Universal Robots PolyScope program: speedSliderEx_wInput.urp

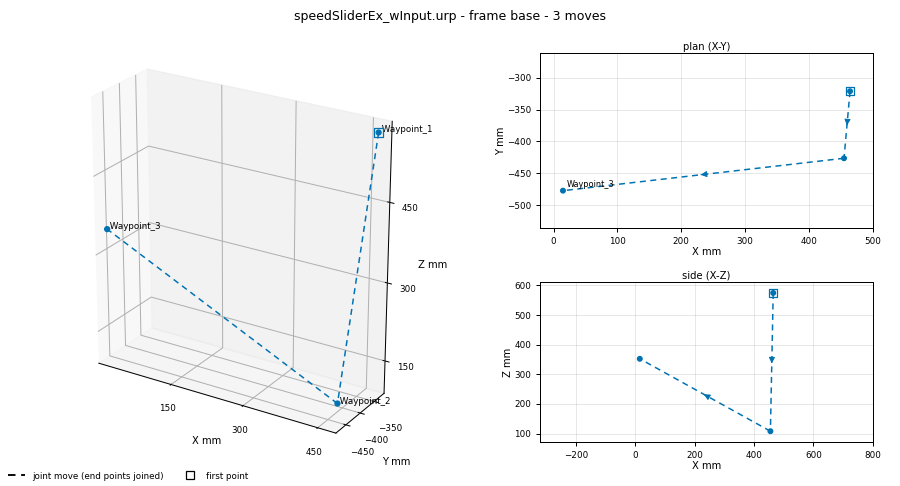
[picture p0: tool path of speedSliderEx_wInput.urp in frame base, 3 of 3 moves have a stored position in this frame; points joined in program order, loops and branches not executed]
ProgramRoot directory=/programs; kinematics=(a=[0, -0.425, -0.39225, 0, 0, 0], d=[0.08916, 0, 0, 0.10915, 0.09465, 0.0823], alpha=[1.5708, 0, 0, 1.5708, -1.5708, 0], deltaTheta=[0, 0, 0, 0, 0, 0], status=notInitialized); name=speedSliderEx_wInput; programVersion=(project__name=PolyScope, major__version=1, minor__version=8, svn__revision=14035, build__date=Apr 28 2014, 10:06:36); robotEnvironmentFileName=default; serialNumberRobot=2012209394
  MainProgram cartesianAcceleration=1.2; cartesianSpeed=12.0; jointAcceleration=1.3962634015954636; jointSpeed=1.0471975511965976; moveAsFastAsPossible=true; sharedProcessMoveBlendRadius=0.025; featureReference=(installationNameReference=Base); motionType=JOINT_SPACE
    Move cartesianAcceleration=1.2; cartesianSpeed=12.0; jointAcceleration=1.3962634015954636; jointSpeed=1.0471975511965976; moveAsFastAsPossible=true; sharedProcessMoveBlendRadius=0.025; featureReference=(installationNameReference=Base); motionType=JOINT_SPACE
      Waypoint blendRadius=0.05; cartesianAcceleration=1.2; cartesianSpeed=12.0; jointAcceleration=1.3962634015954636; jointSpeed=1.0471975511965976; nextMotionTime=2.0; stoppoint=true; useSharedBlendParameter=true; useSharedParameters=true; position=TCP in base x=464.486 y=-321.339 z=574.383 mm, rx=2.3556 ry=2.0077 rz=0.0323 rad; joints [-23.52, -102.508, -55.368, -109.215, 89.91, -194.406] deg; positionType=FIXED_POSITION; waypointPoseInFeatureCoordinates=(pos=(x=0.4644861952459154, y=-0.32133933165581147, z=0.5743832469432477), rot=(x=2.3556191427131474, y=2.0077422491662906, z=0.03225842255249453)); name=Waypoint_1
      Waypoint blendRadius=0.05; cartesianAcceleration=1.2; cartesianSpeed=12.0; jointAcceleration=1.3962634015954636; jointSpeed=1.0471975511965976; nextMotionTime=2.0; stoppoint=true; useSharedBlendParameter=true; useSharedParameters=true; position=TCP in base x=455.044 y=-426.389 z=108.273 mm, rx=2.4747 ry=1.777 rz=0.0523 rad; joints [-33.038, -122.072, -101.148, -41.016, 89.865, -194.406] deg; positionType=FIXED_POSITION; waypointPoseInFeatureCoordinates=(pos=(x=0.45504385007230075, y=-0.42638941830143984, z=0.1082728784381753), rot=(x=2.4747428751253917, y=1.7769546800298406, z=0.052269962504872085)); name=Waypoint_2
      Waypoint blendRadius=0.05; cartesianAcceleration=1.2; cartesianSpeed=12.0; jointAcceleration=1.3962634015954636; jointSpeed=1.0471975511965976; nextMotionTime=2.0; stoppoint=true; useSharedBlendParameter=true; useSharedParameters=true; position=TCP in base x=14.703 y=-477.16 z=352.369 mm, rx=-2.9182 ry=-0.7779 rz=0.053 rad; joints [-74.672, -89.173, -100.903, -86.873, 88.044, -194.406] deg; positionType=FIXED_POSITION; waypointPoseInFeatureCoordinates=(pos=(x=0.014702750511910391, y=-0.47715952925743804, z=0.3523688298737984), rot=(x=-2.918194551957495, y=-0.7779111021492721, z=0.053016427281325745)); name=Waypoint_3
  Thread name=Thread_1
    Assignment assignmentValueSource=0; expr=socket_open("127.0.0.1", 30002); operatorValueType=INTEGER; valueSource=EXPRESSION; variable=(name=ok, prefersPersistentValue=false, requestANewUniqueName=false)
    Assignment assignmentValueSource=0; expr=0.2; operatorValueType=INTEGER; valueSource=EXPRESSION; variable=(name=speed_low, prefersPersistentValue=false, requestANewUniqueName=false)
    Assignment assignmentValueSource=0; expr=1.0; operatorValueType=INTEGER; valueSource=EXPRESSION; variable=(name=speed_high, prefersPersistentValue=false, requestANewUniqueName=false)
    While count=0; type=LOOP_FOREVER; variable=(name=Loop_4, prefersPersistentValue=false, requestANewUniqueName=false)
      If expr=digital_in[0] ≟ False; type=IF_NODE
        Assignment assignmentValueSource=0; expr=ExpressionVariableNode; operatorValueType=INTEGER; valueSource=EXPRESSION; variable=(name=speed, prefersPersistentValue=false, requestANewUniqueName=false)
      If type=ELSE_NODE
        Assignment assignmentValueSource=0; expr=ExpressionVariableNode; operatorValueType=INTEGER; valueSource=EXPRESSION; variable=(name=speed, prefersPersistentValue=false, requestANewUniqueName=false)
      Script type=0; expressionBranchNode=socket_send_string("set speed")
      Script type=0; expressionBranchNode=socket_send_string(ExpressionVariableNode)
      Script type=0; expressionBranchNode=socket_send_byte(10)
      Assignment assignmentValueSource=0; expr=digital_in[0]; operatorValueType=INTEGER; valueSource=EXPRESSION; variable=(name=btnState, prefersPersistentValue=false, requestANewUniqueName=false)
      Wait analogComparison=0; analogInputRange=0; analogValue=0.0; digitalValue=0; selectedAnalogSensor=-1; selectedDigitalSensor=-1; waitTime=0.01; expr=ExpressionVariableNode≠ digital_in[0]; type=EXPRESSION_WAIT
